// Mitsubishi GX Works2 project: 산업기사공개문제   PLC: Q02/Q02H

PROGRAM MAIN
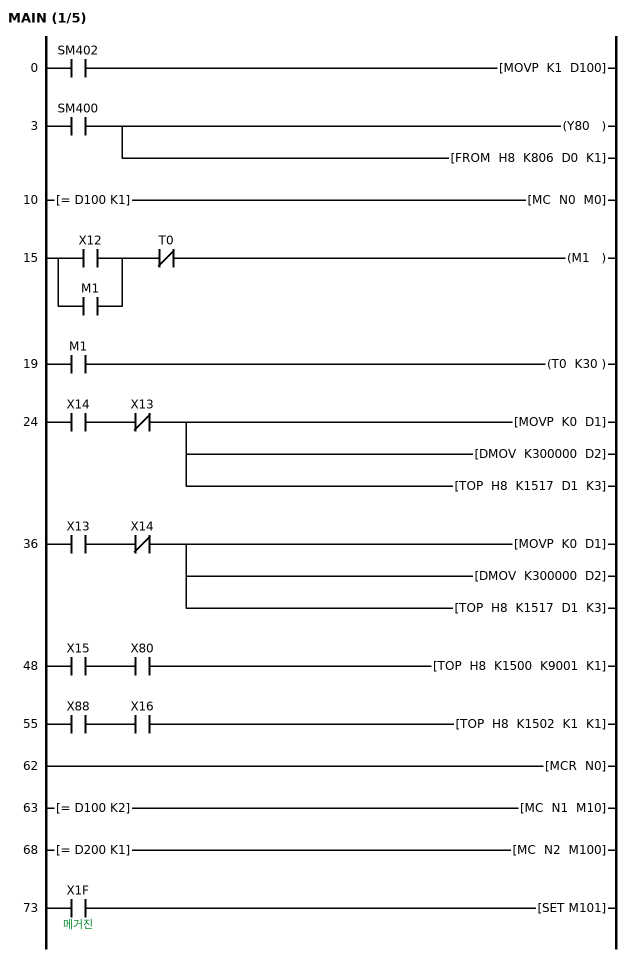
0     LD      SM402
      MOVP    K1 D100
3     LD      SM400
      OUT     Y80
      FROM    H8 K806 D0 K1
10    LD=     D100 K1
      MC      N0 M0
15    LD      X12
      OR      M1
      ANI     T0
      OUT     M1
19    LD      M1
      OUT     T0 K30
24    LD      X14
      ANI     X13
      MOVP    K0 D1
      DMOV    K300000 D2
      TOP     H8 K1517 D1 K3
36    LD      X13
      ANI     X14
      MOVP    K0 D1
      DMOV    K300000 D2
      TOP     H8 K1517 D1 K3
48    LD      X15
      AND     X80
      TOP     H8 K1500 K9001 K1
55    LD      X88
      AND     X16
      TOP     H8 K1502 K1 K1
62    MCR     N0
63    LD=     D100 K2
      MC      N1 M10
68    LD=     D200 K1
      MC      N2 M100
73    LD      X1F  ; 메거진
      SET     M101
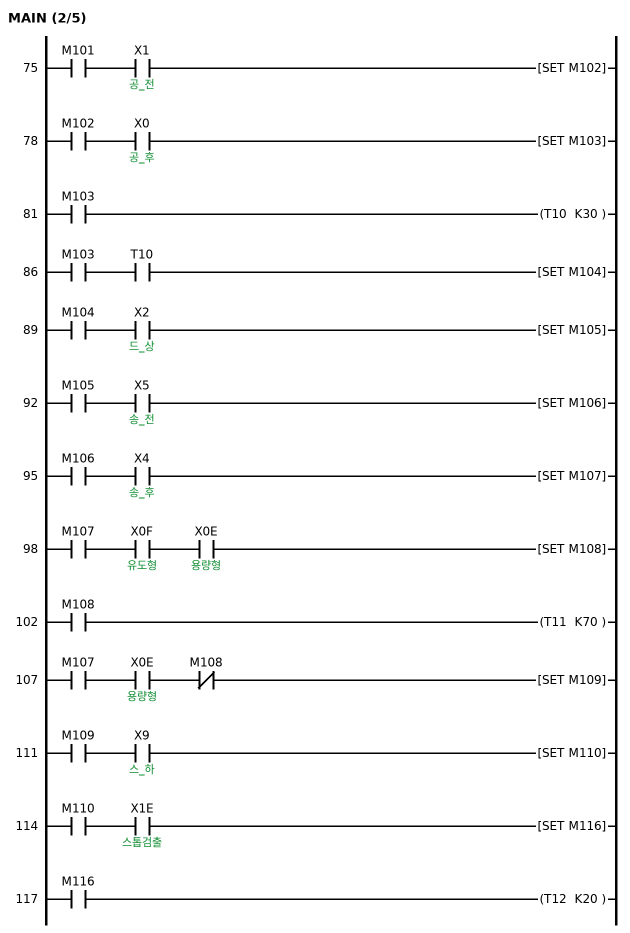
75    LD      M101
      AND     X1  ; 공_전
      SET     M102
78    LD      M102
      AND     X0  ; 공_후
      SET     M103
81    LD      M103
      OUT     T10 K30
86    LD      M103
      AND     T10
      SET     M104
89    LD      M104
      AND     X2  ; 드_상
      SET     M105
92    LD      M105
      AND     X5  ; 송_전
      SET     M106
95    LD      M106
      AND     X4  ; 송_후
      SET     M107
98    LD      M107
      AND     X0F  ; 유도형
      AND     X0E  ; 용량형
      SET     M108
102   LD      M108
      OUT     T11 K70
107   LD      M107
      AND     X0E  ; 용량형
      ANI     M108
      SET     M109
111   LD      M109
      AND     X9  ; 스_하
      SET     M110
114   LD      M110
      AND     X1E  ; 스톱검출
      SET     M116
117   LD      M116
      OUT     T12 K20
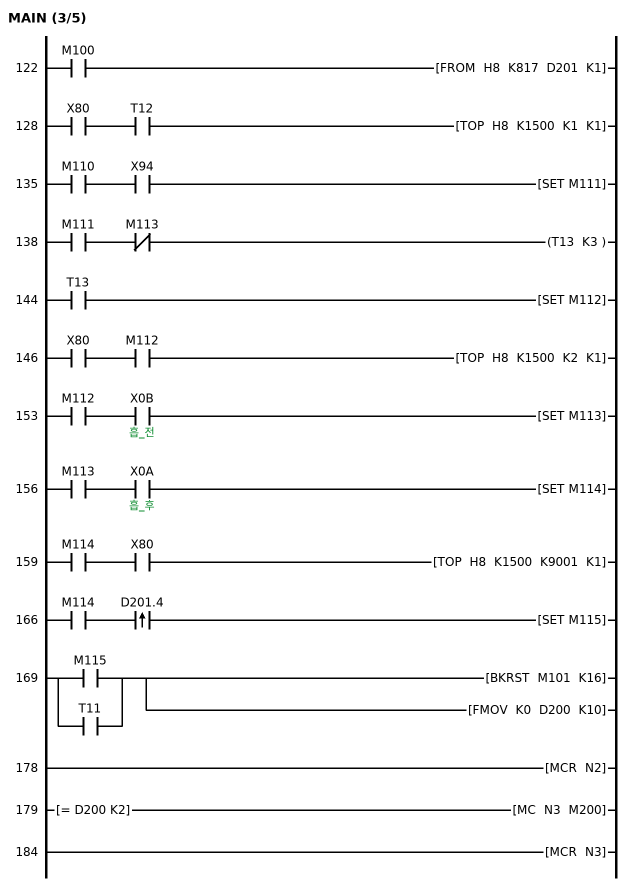
122   LD      M100
      FROM    H8 K817 D201 K1
128   LD      X80
      AND     T12
      TOP     H8 K1500 K1 K1
135   LD      M110
      AND     X94
      SET     M111
138   LD      M111
      ANI     M113
      OUT     T13 K3
144   LD      T13
      SET     M112
146   LD      X80
      AND     M112
      TOP     H8 K1500 K2 K1
153   LD      M112
      AND     X0B  ; 흡_전
      SET     M113
156   LD      M113
      AND     X0A  ; 흡_후
      SET     M114
159   LD      M114
      AND     X80
      TOP     H8 K1500 K9001 K1
166   LD      M114
      ANDP    D201.4
      SET     M115
169   LD      M115
      OR      T11
      BKRST   M101 K16
      FMOV    K0 D200 K10
178   MCR     N2
179   LD=     D200 K2
      MC      N3 M200
184   MCR     N3
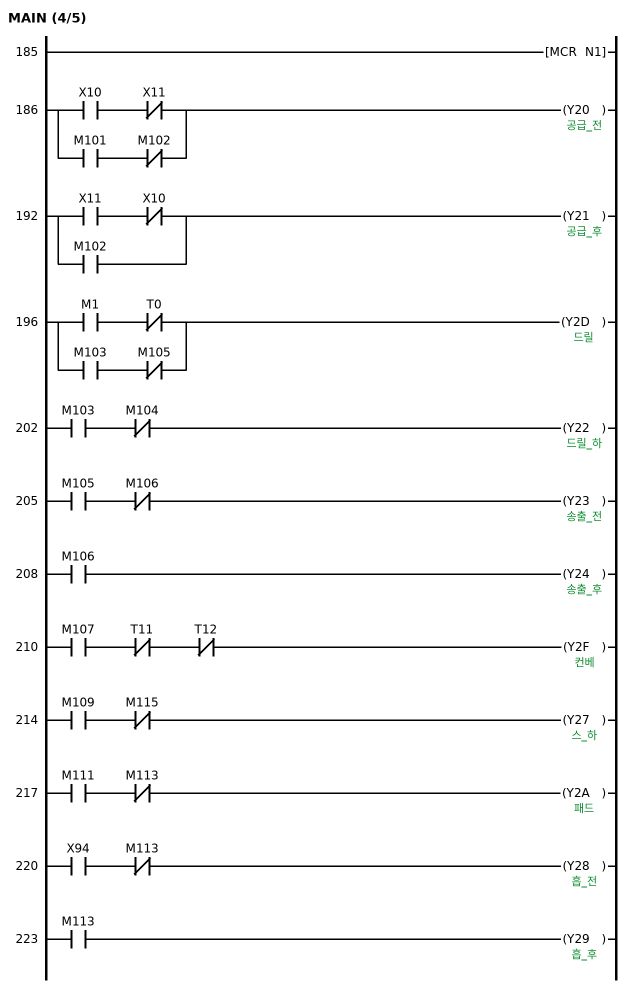
185   MCR     N1
186   LD      X10
      ANI     X11
      LD      M101
      ANI     M102
      ORB
      OUT     Y20  ; 공급_전
192   LD      X11
      ANI     X10
      OR      M102
      OUT     Y21  ; 공급_후
196   LD      M1
      ANI     T0
      LD      M103
      ANI     M105
      ORB
      OUT     Y2D  ; 드릴
202   LD      M103
      ANI     M104
      OUT     Y22  ; 드릴_하
205   LD      M105
      ANI     M106
      OUT     Y23  ; 송출_전
208   LD      M106
      OUT     Y24  ; 송출_후
210   LD      M107
      ANI     T11
      ANI     T12
      OUT     Y2F  ; 컨베
214   LD      M109
      ANI     M115
      OUT     Y27  ; 스_하
217   LD      M111
      ANI     M113
      OUT     Y2A  ; 패드
220   LD      X94
      ANI     M113
      OUT     Y28  ; 흡_전
223   LD      M113
      OUT     Y29  ; 흡_후
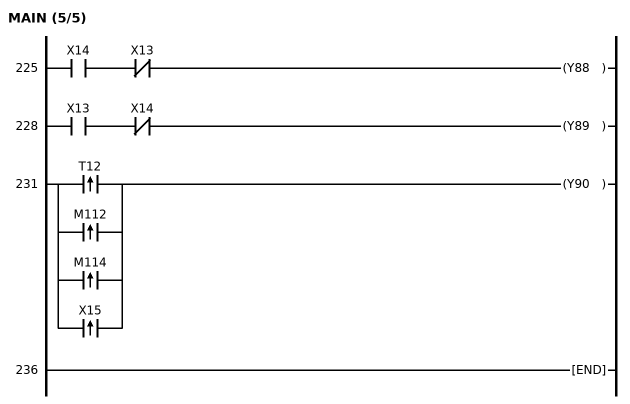
225   LD      X14
      ANI     X13
      OUT     Y88
228   LD      X13
      ANI     X14
      OUT     Y89
231   LDP     T12
      ORP     M112
      ORP     M114
      ORP     X15
      OUT     Y90
236   END
END_PROGRAM

// device comments not shown above
X3  ; 드_하
X6  ; 배_후
X7  ; 배_전
X8  ; 스_상
X0C  ; 창_후
X0D  ; 창_전
Y25  ; 배출_전
Y26  ; 배출_후
Y2B  ; 창전
Y2C  ; 창후
